{attribute 'qualified_only'}
{attribute 'strict'}
{attribute 'to_string'}
TYPE E_BridgeStatus :
(
    Connected,
    LocalNotOperational,
    RemoteNotConnected,
    RemoteNotOperational,
    LinkError,
    DataStale
) UDINT;
END_TYPE

(* stored: Version 1.1.0.1, ProductVersion 3.1.4024.12
   DUT E_BridgeStatus: Id {5d6adaaf-7075-438d-856d-a489d0a9a0c4} *)
